LIN {X 0,Y 164.296,Z 431.128,A -85,B 0,C 180,E1 -31511.938,E2 -31511.938} C_VEL
LIN {X 0,Y 165.59,Z 423.848,A -85,B 0,C 180,E1 -31511.971,E2 -31511.971} C_VEL
LIN {X 0,Y 165.554,Z 423.773,A -85,B 0,C 180,E1 -31514.19,E2 -31514.19} C_VEL
LIN {X 0,Y 165.491,Z 424.37,A -85,B 0,C 180,E1 -31515.36,E2 -31515.36} C_VEL
LIN {X 0,Y 163.75,Z 433.674,A -85,B 0,C 180,E1 -31515.428,E2 -31515.428} C_VEL
LIN {X 0,Y 163.707,Z 434.103,A -85,B 0,C 180,E1 -31515.434,E2 -31515.434} C_VEL
LIN {X 0,Y 163.707,Z 600,A -85,B 0,C 180,E1 -31515.434,E2 -31515.434} C_VEL
LIN {X 0,Y 163.707,Z 600,A -85,B 0,C 180,E1 -31515.434,E2 -31515.434}

QRS_NEXT_CUT()

QRS_NEXT()
QRS_HOME()

END
